// TwinCAT 3 PLC project IotMqttSampleAzureIotHubDeviceTwin
// ProgramVersion: 3.1.4021.2
// libraries:
//   Tc2_Standard, * (Beckhoff Automation GmbH)
//   Tc2_System, * (Beckhoff Automation GmbH)
//   Tc2_Utilities, * (Beckhoff Automation GmbH)
//   Tc3_IotBase, * (Beckhoff Automation GmbH)
//   Tc3_JsonXml, * (Beckhoff Automation GmbH)
//   Tc3_Module, * (Beckhoff Automation GmbH)
// project tree:
//   / PlcTask.TcTTO
//   POUs/ FB_TopicInfos.TcPOU, MAIN.TcPOU, F_GetTopicInfos.TcPOU, PrgMqttCom.TcPOU
// real-time tasks:
//   TASK PlcTask: cycle T#10ms, priority 20, ADS port 350

CONFIGURATION IotMqttSampleAzureIotHubDeviceTwin
    RESOURCE PLC ON TwinCAT3
        TASK PlcTask(INTERVAL := T#10ms, PRIORITY := 20);
        PROGRAM MAIN WITH PlcTask : MAIN;
    END_RESOURCE
END_CONFIGURATION

// ---- POUs/MAIN.TcPOU
PROGRAM MAIN
VAR
	n : INT;
END_VAR

n := n + 1;

PrgMqttCom();

END_PROGRAM

// ---- POUs/PrgMqttCom.TcPOU
PROGRAM PrgMqttCom
VAR
	fbMqttClient : FB_IotMqttClient;
	fbMessageQueue : FB_IotMqttMessageQueue;
	fbMessage : FB_IotMqttMessage;
	hrErrorOccurred : HRESULT; // contains the latest occurred error
	bSetParameter : BOOL := TRUE;
	bConnect : BOOL := TRUE;
	fbGetTime : GETSYSTEMTIME;
	ftTemp : T_FileTime;
	dtTimestamp : DT;
	
	(* Topic parsing *)
	fbTopicInfos : FB_TopicInfos();
	
	(* IoT Hub Telemetry Data *)
	sTopicTelemtry : STRING(255) := 'devices/CX-12345/messages/events/readpipe/'; // Insert correct DeviceId
	sTopicCloud2Device : STRING(255) := 'devices/CX-12345/messages/devicebound/#'; // Insert correct DeviceId
	sTelemetryData : STRING(2000);
	bSubscribed : BOOL; // Indicates that the MQTT driver has successfully subscribed to the Cloud2Device topic	
	i: UDINT;
	fbTimer : TON := (PT:=T#1S); // timer to send telemetry data
	{attribute 'TcEncoding':='UTF-8'}
	sTopicRcv : STRING(255);
	{attribute 'TcEncoding':='UTF-8'}
	sCloud2DeviceMessage : STRING(255);
	
	(* Device Twin topics *)
	sTopicTwinResponses : STRING(255) := '$$iothub/twin/res/#';
	sTopicTwinGetBase : STRING(255) := '$$iothub/twin/GET/?$$rid=';
	sTopicTwinUpdateBase : STRING(255) := '$$iothub/twin/PATCH/properties/reported/?$$rid=';
	sTopicTwinDesired : STRING(255) := '$$iothub/twin/PATCH/properties/desired/#';
	sTopicTwinMethodsPost : STRING(255) := '$$iothub/methods/POST/#';
	sTopicTwinMethodsResBase : STRING(255) := '$$iothub/methods/res/'; 
	sTopicTwinMethodsResActual : STRING(255) := '';
	sTopicTwinGetActual : STRING(255);
	sTopicTwinUpdateActual : STRING(255);
	sTopicInfos : STRING(255);
	
	(* Device Twin method call *)
	sTwinMethodCallName : STRING(255);
	sTwinMethodCallId : STRING(255);
	sTwinMethodCallContent : STRING(255);
	
	(* Device Twin response *)
	sTwinResponse : STRING(255);
	
	(* Device Twin actions and trigger *)
	bTwinGet : BOOL := FALSE; // Receives the current Device Twin document (received in sTwinResponse)
	bTwinUpdate : BOOL := FALSE; // Starts an UPDATE operation on the Device Twin
	bTwinDeleteProperty : BOOL := FALSE; // Deletes a property from the Device Twin
	bTwinMethodCallReceived : BOOL := FALSE; // Indicates that a MethodCall has been received by the Device Twin
	bTwinSubscribed : BOOL := FALSE; // Indicates that the MQTT driver has successfully subscribed to the Device Twin Response topic
	bTwinDesiredSubscribed : BOOL := FALSE; // Indicates that the MQTT driver has successfully subscribed to the Device Twin Desired topic
	bTwinMethodsPostSubscribed : BOOL := FALSE; // Indicates that the MQTT driver has successfully subscribed to the Device Twin MethodCall topic
	
	(* Temporary variables to either GET or UPDATE the Device Twin *)
	sJsonTwinGet : STRING(0); // Empty content to receive Device Twin document
	sJsonTwinUpdate : STRING(255); // Stores updates for the Device Twin
	
	nTwinRequestId : UINT := 1;
	nResStatusCode : UDINT;
	nResRequestId : UDINT;
	
	(* JSON parsing *)
	fbJson      : FB_JsonSaxWriter;
	fbJsonTwinUpdate : FB_JsonSaxWriter;

END_VAR

IF bSetParameter THEN
	bSetParameter := FALSE;
	fbMqttClient.stTLS.sCA := 'c:\TwinCAT\3.1\Config\Certificates\Azure\BaltimoreRoot.cer'; // CA certificate 
	fbMqttClient.stTLS.sAzureSas := 'HostName=beckhoff-automation.azure-devices.net;DeviceId=CX-12345;SharedAccessSignature=SharedAccessSignature sr=beckhoff-automation.azure-devices.net%2Fdevices%2FCX-12345&sig=PHAG36uxZw9s1przM25YmwViKIG6twB0YSEUW45xJDk%3D&se=1613540738'; // Device SAS Token
	fbMqttClient.ipMessageQueue := fbMessageQueue;
END_IF

fbMqttClient.Execute(bConnect);
IF fbMqttClient.bError THEN
	// add your error logging here
	hrErrorOccurred := fbMqttClient.hrErrorCode;
END_IF

(* Check for received messages and parse them *)
IF fbMessageQueue.nQueuedMessages > 0 THEN
	IF fbMessageQueue.Dequeue(fbMessage:=fbMessage) THEN
		fbMessage.GetTopic(pTopic:=ADR(sTopicRcv), nTopicSize:=SIZEOF(sTopicRcv));
		fbTopicInfos(sTopic := sTopicRcv);
		IF fbTopicInfos.IsSystemTopic() THEN
			(* Message comes from one of the system topics - now check which one (Methods or Twin) *)
			IF fbTopicInfos.IsMethodCallTopic() THEN
				(* Message is an incoming method call -> extract MethodName, MethodId and MethodContent *)
				(* MethodName and MethodId are part of the topic, MethodContent is in message payload *)
				bTwinMethodCallReceived := TRUE;
				fbMessage.GetPayload(pPayload:=ADR(sTwinMethodCallContent), nPayloadSize:=SIZEOF(sTwinMethodCallContent), bSetNullTermination:=TRUE);
			ELSE
				(* Message is a regular response -> extract StatusCode and RequestId *)
				(* StatusCode and RequestId are part of the topic *)				
				IF fbTopicInfos.StatusCode <> 200 THEN
					// request wasn't successful - do something
					;
				END_IF
				fbMessage.GetPayload(pPayload:=ADR(sTwinResponse), nPayloadSize:=SIZEOF(sTwinResponse), bSetNullTermination:=TRUE);					
			END_IF
		ELSE
			(* Message is a Cloud2Device message *)
			fbMessage.GetPayload(pPayload:=ADR(sCloud2DeviceMessage), nPayloadSize:=SIZEOF(sCloud2DeviceMessage), bSetNullTermination:=TRUE);
		END_IF
	END_IF
END_IF

IF fbMqttClient.bConnected THEN

	(* Subscribe to all required Device Twin topics *)
	IF NOT bSubscribed THEN
		bSubscribed := fbMqttClient.Subscribe(sTopic:=sTopicCloud2Device, eQoS:=TcIotMqttQos.AtLeastOnceDelivery);
	END_IF
	IF NOT bTwinSubscribed THEN
		bTwinSubscribed := fbMqttClient.Subscribe(sTopic:=sTopicTwinResponses, eQoS:=TcIotMqttQos.AtLeastOnceDelivery);
	END_IF
	IF NOT bTwinDesiredSubscribed THEN
		bTwinDesiredSubscribed := fbMqttClient.Subscribe(sTopic:=sTopicTwinDesired, eQoS:=TcIotMqttQos.AtLeastOnceDelivery);
	END_IF
	IF NOT bTwinMethodsPostSubscribed THEN
		bTwinMethodsPostSubscribed := fbMqttClient.Subscribe(sTopic:=sTopicTwinMethodsPost, eQoS:=TcIotMqttQos.AtLeastOnceDelivery);
	END_IF

	(* Receives the Device Twin document *)
	IF bTwinGet THEN
		bTwinGet := FALSE;
		sTopicTwinGetActual := CONCAT(sTopicTwinGetBase, UINT_TO_STRING(nTwinRequestId));
		nTwinRequestId := nTwinRequestId + 1;
		fbMqttClient.Publish(	sTopic:= sTopicTwinGetActual, 
								pPayload:= ADR(sJsonTwinGet), nPayloadSize:= 0, 
								eQoS:= TcIotMqttQos.AtMostOnceDelivery, bRetain:= FALSE, bQueue:= FALSE );		
	END_IF
	
	(* Updates the Device Twin document *)
	IF bTwinUpdate THEN
		bTwinUpdate := FALSE;
		sTopicTwinUpdateActual := CONCAT(sTopicTwinUpdateBase, UINT_TO_STRING(nTwinRequestId));
		nTwinRequestId := nTwinRequestId + 1;			
		fbJsonTwinUpdate.StartObject();
		fbJsonTwinUpdate.AddKey('OperatingSystem');
		fbJsonTwinUpdate.AddString('Windows 10 IoT Enterprise');
		fbJsonTwinUpdate.AddKey('Hostname');
		fbJsonTwinUpdate.AddString('CX-12345');
		fbJsonTwinUpdate.AddKey('TwinCatVersion');
		fbJsonTwinUpdate.AddString('3.1 Build 4024.7');		
		fbJsonTwinUpdate.EndObject();
		sJsonTwinUpdate := fbJsonTwinUpdate.GetDocument();
		fbJsonTwinUpdate.ResetDocument();
		fbMqttClient.Publish(	sTopic:= sTopicTwinUpdateActual, 
								pPayload:= ADR(sJsonTwinUpdate), nPayloadSize:= LEN2(ADR(sJsonTwinUpdate)), 
								eQoS:= TcIotMqttQos.AtMostOnceDelivery, bRetain:= FALSE, bQueue:= FALSE );		
	END_IF
	
	(* Removes a property from the Device Twin *)
	IF bTwinDeleteProperty THEN
		bTwinDeleteProperty := FALSE;
		sTopicTwinUpdateActual := CONCAT(sTopicTwinUpdateBase, UINT_TO_STRING(nTwinRequestId));
		nTwinRequestId := nTwinRequestId + 1;
		fbJsonTwinUpdate.StartObject();
		fbJsonTwinUpdate.AddKey('TwinCatVersion');
		fbJsonTwinUpdate.AddNull();		
		fbJsonTwinUpdate.EndObject();
		sJsonTwinUpdate := fbJsonTwinUpdate.GetDocument();
		fbJsonTwinUpdate.ResetDocument();
		fbMqttClient.Publish(	sTopic:= sTopicTwinUpdateActual, 
								pPayload:= ADR(sJsonTwinUpdate), nPayloadSize:= LEN2(ADR(sJsonTwinUpdate)), 
								eQoS:= TcIotMqttQos.AtMostOnceDelivery, bRetain:= FALSE, bQueue:= FALSE );		
	END_IF
	
	(* Incoming method call detected *)
	IF bTwinMethodCallReceived THEN
		IF fbTopicInfos.MethodName = 'MethodName' THEN
			// Method "MethodName" has been called - do something and send response
			// In this example, the response always contains the current telemtry message
			;
		END_IF
		sTopicTwinMethodsResActual := CONCAT(sTopicTwinMethodsResBase, '0'); // Return StatusCode of method call- always '0' in this sample
		sTopicTwinMethodsResActual := CONCAT(sTopicTwinMethodsResActual, '/?');
		sTopicTwinMethodsResActual := CONCAT(sTopicTwinMethodsResActual, '$$rid=');
		sTopicTwinMethodsResActual := CONCAT(sTopicTwinMethodsResActual, fbTopicInfos.MethodID); // MethodCallId
		fbMqttClient.Publish(	sTopic:= sTopicTwinMethodsResActual, 
						pPayload:= ADR(sTelemetryData), nPayloadSize:= LEN2(ADR(sTelemetryData)), 
						eQoS:= TcIotMqttQos.AtMostOnceDelivery, bRetain:= FALSE, bQueue:= FALSE );
		bTwinMethodCallReceived := FALSE;
		sTopicTwinMethodsResActual := '';
	END_IF
	
	fbTimer(IN:=TRUE);
	IF fbTimer.Q THEN // publish new payload every second
		fbTimer(IN:=FALSE);
		i := i + 1;

		(* Generate timestamp *)
		fbGetTime(timeLoDW => ftTemp.dwLowDateTime, timeHiDW => ftTemp.dwHighDateTime);
		dtTimestamp := FILETIME_TO_DT(ftTemp);
		
		(* JSON document is created here *)				
		fbJson.StartObject();
		fbJson.AddKey('Timestamp');
		fbJson.AddDateTime(dtTimestamp);
		fbJson.AddKey('Sensor1');
		fbJson.AddReal(42.42);
		fbJson.AddKey('Sensor2');
		fbJson.AddDint(42);
		fbJson.AddKey('Sensor3');
		fbJson.AddBool(TRUE);
		fbJson.EndObject();
		sTelemetryData := fbJson.GetDocument();
		fbJson.ResetDocument();
		
		fbMqttClient.Publish(	sTopic:= sTopicTelemtry, 
								pPayload:= ADR(sTelemetryData), nPayloadSize:= LEN2(ADR(sTelemetryData)), 
								eQoS:= TcIotMqttQos.AtMostOnceDelivery, bRetain:= FALSE, bQueue:= FALSE );
								
		IF fbMqttClient.bError THEN
			// add your error logging here
			hrErrorOccurred := fbMqttClient.hrErrorCode;
		END_IF
	END_IF
END_IF

END_PROGRAM

// ---- POUs/FB_TopicInfos.TcPOU
FUNCTION_BLOCK FB_TopicInfos
VAR_INPUT
	sTopic : STRING(255);
END_VAR
VAR_OUTPUT
END_VAR
VAR
	bIsMethodCallTopic : BOOL;
	bIsSystemTopic : BOOL;
	bIsTwinTopic : BOOL;
	
	sMethodID : STRING(255);
	sMethodName : STRING(255);
	nRequestID : UINT;
	nStatusCode : UINT;
	
	nTopicLength : UDINT;
	nSubTopicLength : UDINT;
	nMethodsPos : INT;
	nPos : INT;
	
	sTopicParser_1 : STRING;
	sTopicParser_2 : STRING;
	sTopicParser_3 : STRING;
	sTopicParser_4 : STRING;
	sTopicParser_5 : STRING;
END_VAR

bIsSystemTopic := FALSE;
bIsMethodCallTopic := FALSE;
bIsTwinTopic := FALSE;

sTopicParser_1 := LEFT(sTopic, 7);
nTopicLength := LEN2(ADR(sTopic));
IF sTopicParser_1 = '$$iothub' THEN // Device Twin system topic ?
	(* Check if the topic is a MethodCall topic *)
	bIsSystemTopic := TRUE;
	nMethodsPos := FIND(sTopic, 'methods');	
	IF nMethodsPos <> 0 THEN
		bIsMethodCallTopic := TRUE;
		(* format of method topic : $iothub/methods/POST/{method name}/?$rid={request id} *)
		sTopicParser_2 := MID(sTopic, 21, 1); // $$iothub/methods/POST/
		sTopicParser_3 := RIGHT(sTopic, UDINT_TO_INT(nTopicLength - 21)); // {method name}/?$rid={request id}
		nSubTopicLength := LEN2(ADR(sTopicParser_3));
		nPos := FIND(sTopicParser_3, '/');
		sTopicParser_4 := LEFT(sTopicParser_3, nPos - 1); 
		sMethodName := sTopicParser_4;
		nPos := FIND(sTopicParser_3, '=');
		sTopicParser_5 := RIGHT(sTopicParser_3, UDINT_TO_INT(nSubTopicLength - nPos)); 
		sMethodID := sTopicParser_5;
	ELSE
		bIsTwinTopic := TRUE;
		sTopicParser_2 := LEFT(sTopic, 20);
		sTopicParser_3 := RIGHT(sTopicParser_2, 3); // Response status code
		nStatusCode := STRING_TO_UINT(sTopicParser_3);
		sTopicParser_4 := RIGHT(sTopic, UDINT_TO_INT(nTopicLength - 21)); // get last sub-topic
		sTopicParser_5 := MID(sTopicParser_4, UDINT_TO_INT(LEN2(ADR(sTopicParser_4))) - FIND(sTopicParser_4, '='), 7); // retrieve RequestId from response
		nRequestID := STRING_TO_UINT(sTopicParser_5);
	END_IF	
ELSE
	bIsSystemTopic := FALSE;
END_IF

METHOD IsMethodCallTopic : BOOL
VAR_INPUT
END_VAR
IsMethodCallTopic := bIsMethodCallTopic;
END_METHOD

METHOD IsSystemTopic : BOOL
VAR_INPUT
END_VAR
IsSystemTopic := bIsSystemTopic;
END_METHOD

METHOD IsTwinTopic : BOOL
VAR_INPUT
END_VAR
IsTwinTopic := bIsTwinTopic;
END_METHOD

PROPERTY MethodID : STRING(255)
GET
MethodID := sMethodID;
END_GET
END_PROPERTY

PROPERTY MethodName : STRING(255)
GET
MethodName := sMethodName;
END_GET
END_PROPERTY

PROPERTY RequestID : UINT
GET
RequestID := nRequestID;
END_GET
END_PROPERTY

PROPERTY StatusCode : UINT
GET
StatusCode := nStatusCode;
END_GET
END_PROPERTY

END_FUNCTION_BLOCK

// ---- POUs/F_GetTopicInfos.TcPOU
FUNCTION F_GetTopicInfos : STRING(255)
VAR_INPUT
	sTopic : STRING(255);
END_VAR
VAR
	nTopicLength : UDINT;
	nSubTopicLength : UDINT;
	sTopicParser_1 : STRING;
	nMethodsPos : INT;
	nPos : INT;
	sTopicParser_2 : STRING;
	sTopicParser_3 : STRING;
	sTopicParser_4 : STRING;
	sTopicParser_5 : STRING;
	fbJson : FB_JsonSaxWriter;
	nOperationStatusCode : UINT;
	nOperationRequestId : UINT;
END_VAR

sTopicParser_1 := LEFT(sTopic, 7);
nTopicLength := LEN2(ADR(sTopic));
IF sTopicParser_1 = '$$iothub' THEN // Device Twin system topic ?
	(* Check if the topic is a MethodCall topic *)
	nMethodsPos := FIND(sTopic, 'methods');	
	fbJson.StartObject();
	fbJson.AddKey('IsIoTHubSystemTopic');
	fbJson.AddBool(TRUE);
	fbJson.AddKey('IsMethodTopic');
	IF nMethodsPos <> 0 THEN
		fbJson.AddBool(TRUE);
		(* format of method topic : $iothub/methods/POST/{method name}/?$rid={request id} *)
		sTopicParser_2 := MID(sTopic, 21, 1); // $$iothub/methods/POST/
		sTopicParser_3 := RIGHT(sTopic, UDINT_TO_INT(nTopicLength - 21)); // {method name}/?$rid={request id}
		nSubTopicLength := LEN2(ADR(sTopicParser_3));
		nPos := FIND(sTopicParser_3, '/');
		sTopicParser_4 := LEFT(sTopicParser_3, nPos - 1); 
		fbJson.AddKey('MethodName');
		fbJson.AddString(sTopicParser_4);
		fbJson.AddKey('MethodId');
		nPos := FIND(sTopicParser_3, '=');
		sTopicParser_5 := RIGHT(sTopicParser_3, UDINT_TO_INT(nSubTopicLength - nPos)); 
		fbJson.AddString(sTopicParser_5);
	ELSE
		fbJson.AddBool(FALSE);
		sTopicParser_2 := LEFT(sTopic, 20);
		sTopicParser_3 := RIGHT(sTopicParser_2, 3); // Response status code
		nOperationStatusCode := STRING_TO_UINT(sTopicParser_3);
		fbJson.AddKey('StatusCode');
		fbJson.AddDint(nOperationStatusCode);
		sTopicParser_4 := RIGHT(sTopic, UDINT_TO_INT(nTopicLength - 21)); // get last sub-topic
		sTopicParser_5 := MID(sTopicParser_4, UDINT_TO_INT(LEN2(ADR(sTopicParser_4))) - FIND(sTopicParser_4, '='), 7); // retrieve RequestId from response
		nOperationRequestId := STRING_TO_UINT(sTopicParser_5);
		fbJson.AddKey('RequestId');
		fbJson.AddDint(nOperationRequestId);
	END_IF	
	fbJson.EndObject();
	F_GetTopicInfos := fbJson.GetDocument();
	fbJson.ResetDocument();	
END_IF

END_FUNCTION
